Staubli VAL3: DeleteTxt.pgx

program DeleteTxt()
  local num l_nNum
begin


  if libList("Disk://txt",sStrFileName)==false
    return
  endIf

  l_nNum=size(sStrFileName)
  if l_nNum<1
    return
  endIf

  for l_nNum=0 to size(sStrFileName)-1
    if find(sStrFileName[l_nNum],".txt")>0
      $delete("Disk://txt/"+sStrFileName[l_nNum])
    endIf


  endFor





  $fileClose(0)
  $fileClose(1)
  $fileClose(2)
  $fileClose(3)
  $fileClose(4)
  $fileClose(5)
  $fileClose(6)
  $fileClose(7)
  $fileClose(8)
  $fileClose(9)






end
